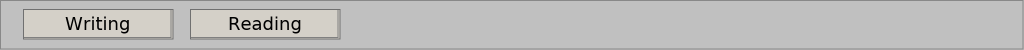
VISUALIZATION Footer  // 1024x50
    Button (23,9 150x30), "Writing"
        OnMouseClick: change screen: Writing
    Button (190,9 150x30), "Reading"
        OnMouseClick: change screen: Reading
END_VISUALIZATION

(* stored: Version 1.1.0.1, ProductVersion 3.1.4024.13
   Visu Footer: Id {87e74a70-60cc-4272-879a-5acaba013ec9} *)
